Staubli VAL3: projetoMiguel.pjx

--- projetoMiguel.pjx ---
Parameters version=s7.11 stackSize=5000 millimeterUnit=true
Program file=start.pgx
Program file=stop.pgx
Program file=trabalhoBatata.pgx
Data file=projetoMiguel.dtx

--- projetoMiguel.dtx ---
dio entradas[4]
  [0] = {link=BasicIO-1\%I0}
  [1] = {link=BasicIO-1\%I1}
  [2] = {link=BasicIO-1\%I2}
  [3] = {link=BasicIO-1\%I3}
dio saida = {link=BasicIO-1\%Q0}
dio start = {link=BasicIO-1\%I5}
dio tipoPar = {link=BasicIO-1\%I4}
jointRs app[12]
  [0] = {j1=27.63, j2=91.42, j3=150, j4=-68.52}
  [1] = {j1=25.45, j2=80.4, j3=150, j4=-58.48}
  [2] = {j1=36.49, j2=61.01, j3=150, j4=-48.6}
  [3] = {j1=14.47, j2=67.84, j3=150, j4=-81.04}
  [4] = {j1=24.89, j2=41.5, j3=150, j4=-65.2}
  [5] = {j1=22.4, j2=33.21, j3=150, j4=-54.34}
  [6] = {j1=-32.67, j2=-10.84, j3=150, j4=-46.58}
  [7] = {j1=-13.08, j2=-54.65, j3=150, j4=-23.02}
  [8] = {j1=-17.29, j2=-60.78, j3=150, j4=-12.02}
  [9] = {j1=-37.18, j2=-56.61, j3=150, j4=-46.27}
  [10] = {j1=-25.4, j2=-76.47, j3=150, j4=-36.63}
  [11] = {j1=-26.05, j2=-89.36, j3=150, j4=-24.77}
jointRs home = {j3=190}
jointRs targets[12]
  [0] = {j1=27.63, j2=91.42, j3=5, j4=-68.52}
  [1] = {j1=25.45, j2=80.4, j3=5, j4=-58.48}
  [2] = {j1=36.49, j2=61.01, j3=5, j4=-48.6}
  [3] = {j1=14.47, j2=67.84, j3=5, j4=-81.04}
  [4] = {j1=24.89, j2=41.5, j3=5, j4=-65.2}
  [5] = {j1=22.4, j2=33.21, j3=5, j4=-54.34}
  [6] = {j1=-32.67, j2=-10.84, j3=5, j4=-46.59}
  [7] = {j1=-13.08, j2=-54.65, j3=5, j4=-23.02}
  [8] = {j1=-17.29, j2=-60.78, j3=5, j4=-12.02}
  [9] = {j1=-37.18, j2=-56.61, j3=5, j4=-46.27}
  [10] = {j1=-25.4, j2=-76.47, j3=5, j4=-36.63}
  [11] = {j1=-26.05, j2=-89.36, j3=5, j4=-24.77}
mdesc mDownSpeed = {accel=23.04, vel=48, decel=23.04}
mdesc mNomSpeed = {accel=25, vel=50, decel=25}
mdesc mUpSpeed = {accel=24.01, vel=49, decel=24.01}
num destino = 3
num origem
tool garra = {fatherId=flange[0], ioLink=valve1}

--- start.pgx ---
program start()
begin
  call trabalhoBatata()
end

--- trabalhoBatata.pgx ---
program trabalhoBatata()
begin
  movej(home,garra,mNomSpeed)
  dioSet(saida,0)
  while true
    if start==false
      if tipoPar==false
        origem=dioGet(entradas)
      else
        destino=dioGet(entradas)
      endIf
    else
      movej(app[origem],garra,mNomSpeed)
      waitEndMove()
      movej(targets[origem],garra,mDownSpeed)
      waitEndMove()
      dioSet(saida,1)
      delay(0.3)
      movej(app[origem],garra,mUpSpeed)
      waitEndMove()
      movej(app[destino],garra,mNomSpeed)
      waitEndMove()
      movej(targets[destino],garra,mDownSpeed)
      waitEndMove()
      dioSet(saida,0)
      delay(0.3)
      movej(app[destino],garra,mUpSpeed)
      waitEndMove()
      movej(home,garra,mNomSpeed)
      waitEndMove()
    endIf
  endWhile
end
